KUKA KRL program: user_sps_ini.src

&ACCESS RV12
&COMMENT user_housekeeping
&USER PKL_AST
DEF user_sps_ini( )
; hier alle User-Aufrufe fuer den SPS.SUB-Ini einpflegen
; insert alle user-funtions for SPS.SUB-Ini





END
